PROGRAM P0_02_AnalogInput
VAR PERSISTENT
	fbMixer_ActualSpeed			:FB_AnalogInput;
	fbMixer_ActualCurrent		:FB_AnalogInput;
	fbSieve_ActualSpeed			:FB_AnalogInput;
	fbChopper_ActualCurrent		:FB_AnalogInput;
	fbSP_ActualPressure			:FB_AnalogInput;
	fbSP_ActualSpeed			:FB_AnalogInput;
	fbSP_WaterTemperature		:FB_TemperatureInput;
	fbSP_LiquidTemperature		:FB_TemperatureInput;
END_VAR

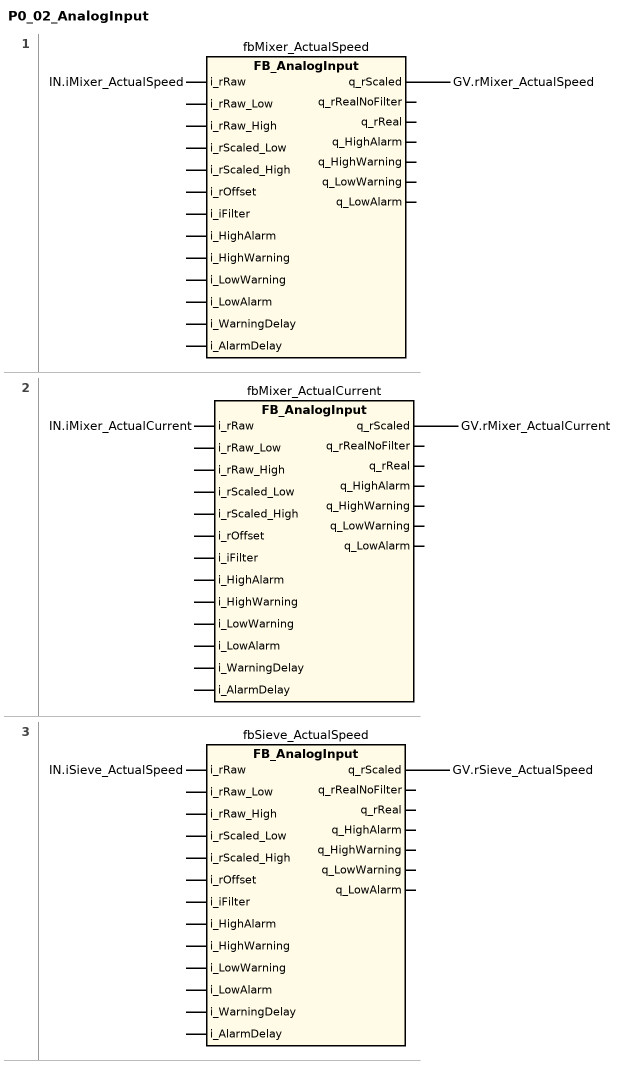
// NETWORK 1
fbMixer_ActualSpeed(i_rRaw := IN.iMixer_ActualSpeed); // FB_AnalogInput
GV.rMixer_ActualSpeed := fbMixer_ActualSpeed.q_rScaled;

// NETWORK 2
fbMixer_ActualCurrent(i_rRaw := IN.iMixer_ActualCurrent); // FB_AnalogInput
GV.rMixer_ActualCurrent := fbMixer_ActualCurrent.q_rScaled;

// NETWORK 3
fbSieve_ActualSpeed(i_rRaw := IN.iSieve_ActualSpeed); // FB_AnalogInput
GV.rSieve_ActualSpeed := fbSieve_ActualSpeed.q_rScaled;

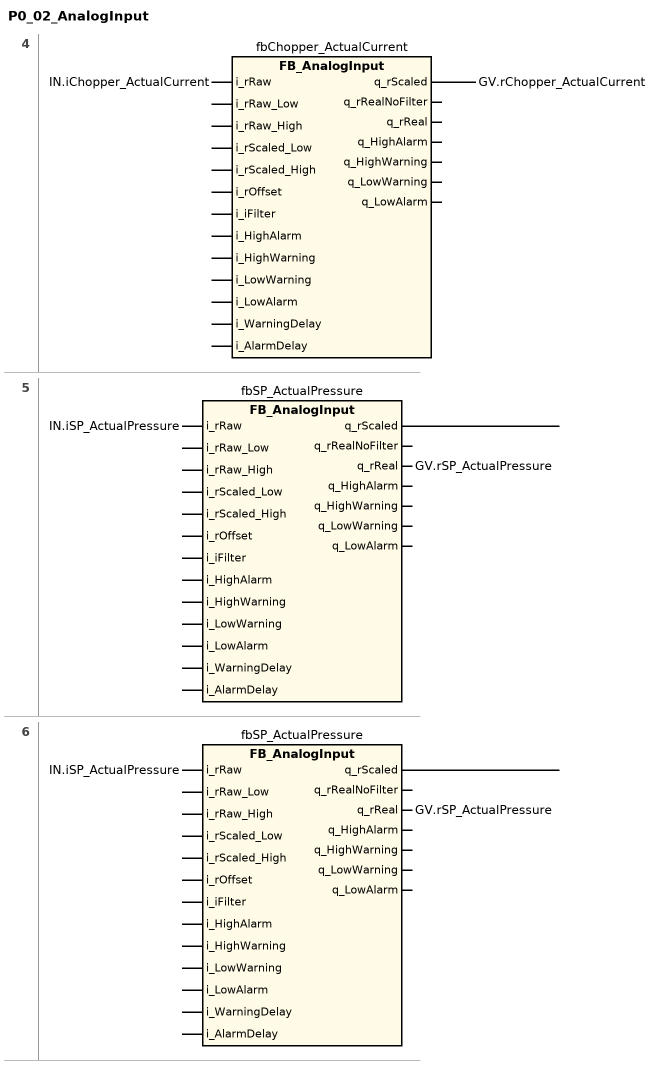
// NETWORK 4
fbChopper_ActualCurrent(i_rRaw := IN.iChopper_ActualCurrent); // FB_AnalogInput
GV.rChopper_ActualCurrent := fbChopper_ActualCurrent.q_rScaled;

// NETWORK 5
fbSP_ActualPressure(i_rRaw := IN.iSP_ActualPressure, q_rReal => GV.rSP_ActualPressure); // FB_AnalogInput

// NETWORK 6
fbSP_ActualPressure(i_rRaw := IN.iSP_ActualPressure, q_rReal => GV.rSP_ActualPressure); // FB_AnalogInput

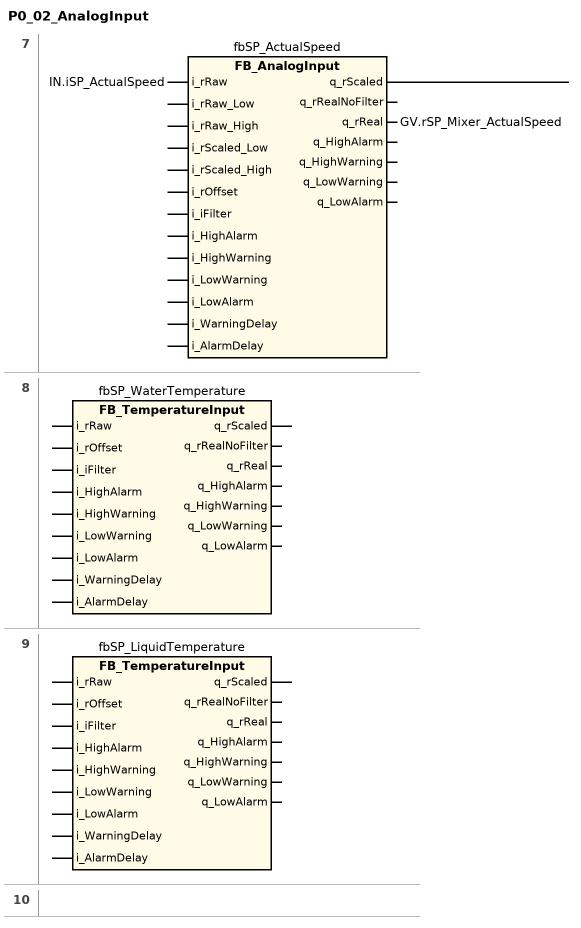
// NETWORK 7
fbSP_ActualSpeed(i_rRaw := IN.iSP_ActualSpeed, q_rReal => GV.rSP_Mixer_ActualSpeed); // FB_AnalogInput

// NETWORK 8
fbSP_WaterTemperature(); // FB_TemperatureInput

// NETWORK 9
fbSP_LiquidTemperature(); // FB_TemperatureInput

// NETWORK 10

END_PROGRAM

(* stored: Version 1.1.0.1, ProductVersion 3.1.4024.12
   POU P0_02_AnalogInput: Id {886e6b80-c86b-4d19-b9e4-45dd208fbc7d}, SpecialFunc None *)
